(* PLC project Generated.project, CODESYS CODESYS V3.5 SP19 Patch 1 *)
(* stored: creationDateTime 2026-09-06T13:00:42.542779, modificationDateTime 2026-09-06T13:00:42.542779 *)

(* ═══════════════════════════════════════════════════════════════ 🕹️ ST_JoystickHMI — Données d'échange IHM pour le Joystick ─────────────────────────────────────────────────────────────── 📄 Structuration en Cmd / State / Cfg , homogène avec ST_ModesHMI. Cfg = réglages FB_Joystick éditables IHM (deadband, temporisations), pontés vers GVL_PERSISTENT via FB_CfgPersistBridge_fbJoystick_Cfg. La calibration du neutre reste dans GVL_PERSISTENT (bouton Calibrate). Pas de Bypass (concept absent de ce struct). ═══════════════════════════════════════════════════════════════ *)
TYPE ST_JoystickHMI : STRUCT
  Cmd : ST_JoystickCmd;
  State : ST_JoystickState;
  Cfg : ST_fbJoystick_Cfg;
END_STRUCT;
END_TYPE

(* ═══════════════════════════════════════════════════════════════ 🎮 ST_JoystickCmd — Commandes IHM pour le Joystick ═══════════════════════════════════════════════════════════════ *)
TYPE ST_JoystickCmd : STRUCT
  Calibrate : BOOL;  (* 🎯 Demande de recalage au neutre (front) *)
END_STRUCT;
END_TYPE

(* ═══════════════════════════════════════════════════════════════ 🚦 ST_JoystickState — États et diagnostics IHM du Joystick ═══════════════════════════════════════════════════════════════ *)
TYPE ST_JoystickState : STRUCT
  RawX : INT;  (* 🕹️ Axe X brut du joystick (0..10000) *)
  RawY : INT;  (* 🕹️ Axe Y brut du joystick (0..10000) *)
  RawButton : BOOL;  (* 🔘 Bouton homme-mort brut *)
  AxisCmdX : ST_fbJoystick_AxisCmd;  (* ⚙️ Consigne d'axe X normalisée (sortie FB_Joystick) *)
  AxisCmdY : ST_fbJoystick_AxisCmd;  (* ⚙️ Consigne d'axe Y normalisée (sortie FB_Joystick) *)
  NeutralXAct : INT;  (* 🎯 Neutre X calibré actuel (lecture seule) *)
  NeutralYAct : INT;  (* 🎯 Neutre Y calibré actuel (lecture seule) *)
  DeadmanArmed : BOOL;  (* 🔫 Geste homme-mort armé (FB_Joystick.DeadmanArmed) *)
  AtNeutral : BOOL;  (* : TRUE si les 2 axes sont en zone morte (position centrale) *)
  Online : BOOL;  (* 📡 Liaison CAN joystick active *)
  Operational : BOOL;  (* 🟢 Joystick opérationnel *)
  Error : BOOL;  (* Joystick en défaut *)
  ErrorId : WORD;  (* ❌ Code défaut joystick *)
END_STRUCT;
END_TYPE

(* ======================================================================= ⚙️ ST_fbJoystick_Cfg — Réglages regroupés de FB_Joystick ─────────────────────────────────────────────────────────────── 🎯 Rôle : porter en un bloc les 5 paramètres de conditionnement du geste (zone morte, temporisations homme-mort, marge défaut capteur). Passé à FB_Joystick via l'entrée `Cfg` — échange bloc IHM / persistant. 🧬 Pattern cfg : aligné sur ST_CycleCfg / ST_WinchCfg (préfixe ST_<Domaine>Cfg, instance persistante dans GVL_PERSISTENT, pont FB_CfgPersistBridge_* à venir). 📄 Doc métier : DOC/AF/AF_Partie-08_Fonction_Joystick_v2.5.md (§5bis) ======================================================================= *)
TYPE ST_fbJoystick_Cfg : STRUCT
  DeadbandRaw : INT := 300;  (* Zone morte en points ADC bruts (0..10000) *)
  NeutralHoldTime : TIME := TIME#100MS;  (* Maintien continu au neutre avant désarmement homme-mort *)
  DeadmanArmHoldTime : TIME := TIME#100MS;  (* Appui continu bouton requis pour armer le geste *)
  DeadmanArmGraceTime : TIME := TIME#3S;  (* Délai de grâce post-armement avant désarmement neutre *)
  RawOutOfRangeMargin : INT := 500;  (* Marge ADC autour des bornes [0..10000] avant défaut capteur (AF08 §5bis) *)
  SpeedStepTable : ST_SpeedStepTable;  (* Les initialiseurs imbriqués de STRUCT (notamment les ARRAY) ne sont pas acceptés par STruCpp/CODESYS dans une déclaration de type. La table est fournie par la configuration persistante de l'appelant. 🪜 Table seuils % -> palier (conversion au joystick, logique FB_Winch §5) *)
  SpeedStepHystMargin : REAL := 2;  (* Marge d'hystérésis palier (%) autour des seuils (anti-oscillation) *)
  Initialized : BOOL := FALSE;  (* 🚦 Flag restauration boot (interne pont FB_CfgPersistBridge_fbJoystick_Cfg) *)
END_STRUCT;
END_TYPE

(* ======================================================================= 🕹️ ST_fbJoystick_AxisCmd — Consigne d'axe normalisée (sortie FB_Joystick) ─────────────────────────────────────────────────────────────── 🎯 Rôle : Structure de consigne d'axe produite par FB_Joystick. 📤 Champs : Enable, StartStop, SpeedTgt (%) + StepTgt (palier 1..5) + direction en bits (DirectionPositive/Negative, AtNeutral). SpeedTgt reste pour l'IHM, StepTgt pour la logique. 📄 Doc métier : DOC/AF/AF_Partie-08_Fonction_Joystick_v2.5.md ======================================================================= *)
TYPE ST_fbJoystick_AxisCmd : STRUCT
  Enable : BOOL;  (* === CONSIGNES DE PILOTAGE AXE === --> [CMD] Autorisation globale pipeline (FALSE=neutralisation, sorties coupees) *)
  StartStop : BOOL;  (* --> [CMD] Validation de mouvement (TRUE=acceleration, FALSE=deceleration/arret) *)
  SpeedTgt : REAL;  (* --> [CMD] Vitesse cible non signee (0...100 %, signe/sens donné par Direction) - IHM *)
  StepTgt : INT;  (* --> [CMD] Palier de vitesse (1..5, 0=arret) - logique/limitations (derive de SpeedTgt) *)
  DirectionNegative : BOOL;  (* --> [CMD] Direction joystick ou intension de gestuelle *)
  DirectionPositive : BOOL;  (* --> [CMD] Direction joystick ou intension de gestuelle *)
  AtNeutral : BOOL;  (* --> [CMD] TRUE si axes en zone morte (position centrale) *)
  Direction : INT;  (* === MONITORING IHM (derive des bits ci-dessus, jamais lu en interlock) === <-- [STAT] Sens -1=Rev / 0=Neutre / +1=Fwd (anim IHM fleche ; lu aussi logique treuils PRG_04) *)
  Deflection : INT;  (* <-- [STAT] Deflexion signee -100..+100 % (anim IHM jauge/barre) *)
END_STRUCT;
END_TYPE

(* ======================================================================= 🪜 ST_SpeedStepTable — Table des paliers de vitesse contacteurs ─────────────────────────────────────────────────────────────── 🎯 Rôle : Structure de configuration des contacteurs et seuils par palier 📄 Doc métier : DOC/AF/AF_Partie-10_Fonction_Winch_v2.1.md ======================================================================= *)
TYPE ST_SpeedStepTable : STRUCT
  P1R1 : BOOL;  (* === PALIER 1 (VITESSE MINIMALE) === Contacteur 1 pour Palier 1 *)
  P1R2 : BOOL;  (* Contacteur 2 pour Palier 1 *)
  P1R3 : BOOL;  (* Contacteur 3 pour Palier 1 *)
  P1R4 : BOOL;  (* Contacteur 4 pour Palier 1 *)
  P2R1 : BOOL;  (* === PALIER 2 === Contacteur 1 pour Palier 2 *)
  P2R2 : BOOL;  (* Contacteur 2 pour Palier 2 *)
  P2R3 : BOOL;  (* Contacteur 3 pour Palier 2 *)
  P2R4 : BOOL;  (* Contacteur 4 pour Palier 2 *)
  P3R1 : BOOL;  (* === PALIER 3 === Contacteur 1 pour Palier 3 *)
  P3R2 : BOOL;  (* Contacteur 2 pour Palier 3 *)
  P3R3 : BOOL;  (* Contacteur 3 pour Palier 3 *)
  P3R4 : BOOL;  (* Contacteur 4 pour Palier 3 *)
  P4R1 : BOOL;  (* === PALIER 4 === Contacteur 1 pour Palier 4 *)
  P4R2 : BOOL;  (* Contacteur 2 pour Palier 4 *)
  P4R3 : BOOL;  (* Contacteur 3 pour Palier 4 *)
  P4R4 : BOOL;  (* Contacteur 4 pour Palier 4 *)
  P5R1 : BOOL;  (* === PALIER 5 (VITESSE MAXIMALE) === Contacteur 1 pour Palier 5 *)
  P5R2 : BOOL;  (* Contacteur 2 pour Palier 5 *)
  P5R3 : BOOL;  (* Contacteur 3 pour Palier 5 *)
  P5R4 : BOOL;  (* Contacteur 4 pour Palier 5 *)
  StepThreshold_Pct : ARRAY[1..5] OF REAL;  (* === SEUILS DE TRANSITION (%) === Seuils de changement de palier (0..100%) *)
END_STRUCT;
END_TYPE
